{attribute 'qualified_only'}
VAR_GLOBAL
	
myPlcAppSystemInfo:PlcAppSystemInfo;
myPlcInfoTask1 : PlcTaskSystemInfo;
myPlcInfoTask2 : PlcTaskSystemInfo;
myPlcInfoTask3 : PlcTaskSystemInfo;
myPlcInfoTask4 : PlcTaskSystemInfo;
myPlcInfoTask5 : PlcTaskSystemInfo;
myPlcInfoTask6 : PlcTaskSystemInfo;


ScanTimeReq:REAL; //the programmed task scan time, e.g. 1, 10, 15, 30ms, etc
ScanTimeAct:REAL; //the last scan time, effective current scan time.

ScanTimeRecord:REAL; //the record scan time
ScanTimeRecordScan:LREAL; //the scan number of the record scan time




END_VAR

(* stored: Version 1.1.0.1, ProductVersion 3.1.4024.12
   GVL System: Id {fa1ba82a-a43b-47a5-9097-4bd33bbfce0d} *)
